// TIA Portal V18 export
DATA_BLOCK "M6doors"   // DB26
VERSION : 0.1
// stored: AutoNumber true, DBAccessibleFromOPCUA true, InstanceOfName axis_FBD, InstanceOfType FB
"axis_FBD"
   // VAR_INPUT
   //    "mm_per_ reductur outputshaft_rev (AskURmechEngineer)" : Real;
   //    "reduction_ rotation (AskURmechEngineer)" : Real;
   //    "ABincrements_per_ encoder_rev (CheckEnc Label and HSC hardware settings dont forget input filtration)" : Real;
   //    "max_revs_ at_10V (CheckMotorLabel)" : Real;
   //    "enc_placed_ on_motor not reductor output shaft(visually inspect)" : Bool;
   //    "isMultiturn (visually inspect)" : Bool;
   //    MultiTurnGoesFwdOnly : Bool;
   //    soft_speed_change_req : Bool;
   //    ENC_REVERSED_DIR : Bool;
   //    ENCODER_DINT : DInt;
   //    TargetUnison : Real;
   //    TargetHome : Real;
   //    Desk_bHome : Bool;
   //    Desk_bFwd : Bool;
   //    Desk_bRev : Bool;
   //    s_fwd_mechOK : Bool;
   //    s_rev_mecOK : Bool;
   //    s_fwd_ind : Bool;
   //    s_rev_ind : Bool;
   //    xPredifCal : Bool;
   //    ALIEN_MODE_EN : Bool;
   //    ALIEN_FWD : Bool;
   //    ALIEN_REV : Bool;
   //    ALIEN_SPDABS : Real;
   //    ExecUni : Bool;
   //    TheseAreDoors : Bool;
   //    xOverrideLocal : Bool;
   //    hbStepPlus : Bool;
   //    hbStepMinus : Bool;
   //    TargetStep : Real;
   //    динамические_границы_используются : Bool;
   //    динамическая_граница_fwd : Real;
   //    динамическая_граница_rev : Real;
   // END_VAR
   // VAR_OUTPUT
   //    max_speed_10V_p_mm : Real;
   //    speed_V : Real;
   //    speed : Real;
   //    yaINTSPEED : Int;
   //    yFWD : Bool;
   //    yREV : Bool;
   //    yFwd_STOP : Bool;
   //    yRev_STOP : Bool;
   //    yIN_POS : Bool;
   //    ER : Bool;
   //    WN : Bool;
   //    ALLOWED : Bool;
   //    "dist_stop(check t_acc)" : Real;
   //    MovingHomeWhileFree : Bool;
   //    ERWSTRING : WString;
   // END_VAR
   // VAR_IN_OUT
   //    aut_target : Real;
   //    para : "typeMotPara";
   //    POS : Real;
   //    calibrated : Bool;
   //    ENC_RET : "typePOSMEMcalib";
   // END_VAR
   // VAR
   //    para_ArtLimits { ExternalAccessible := 'False'; ExternalVisible := 'False'; ExternalWritable := 'False'} : "typeMotPara";
   //    v_absMax : Real;
   //    au_execute : Bool;
   //    AMANGRDB { S7_SetPoint := 'True'} : "axis_manager";
   //    MOTDB { S7_SetPoint := 'True'} : "__mot_universal_";
   //    WNDB { S7_SetPoint := 'True'} : "ER_WORD";
   //    ERDB { S7_SetPoint := 'True'} : "ER_WORD";
   //    erw_calcspd : WString;
   //    hmiResetCalib : Bool;
   //    IEC_Timer_0_Instance { S7_SetPoint := 'True'} : TON_TIME;
   //    artLimiter_Instance { S7_SetPoint := 'True'} : "artLimiter";
   // END_VAR
BEGIN
END_DATA_BLOCK
